// TIA Portal V20 export
// export: Created 2026-04-28T10:05:07.7940218Z, ExportSetting WithDefaults, DisplayName Totally Integrated Automation Portal, DisplayVersion V20, DisplayName TIA Portal Openness, DisplayVersion V20, DisplayName TIA Portal Version Control Interface, DisplayVersion V20, DisplayName SINAMICS Startdrive Advanced, DisplayVersion V20, DisplayName SINAMICS Startdrive G130, G150, S120, S150, SINAMICS MV, G220, S200, S210, DisplayVersion V20, DisplayName SINAMICS Startdrive G110M, G120, G120C, G120D, G120P, G115D, DisplayVersion V20, DisplayName STEP 7 Professional, DisplayVersion V20, DisplayName STEP 7 Safety, DisplayVersion V20, DisplayName WinCC Basic/Comfort/Advanced, DisplayVersion V20, DisplayName WinCC Unified, DisplayVersion V20
TYPE "Daten_SPT_50"
// stored: IsFailsafeCompliant false
   STRUCT
      xMaFa : Bool := false;   // Selection Main fan
      xMaFaSoll : Bool := false;   // Selection Main fan Set Value
      xMaFaIst : Bool := false;   // Selection Main fan Actual Value
      txt_rMoCuMa : DInt := 0;   // Max. motor current, limit
      txt_rMainFanFU : DInt := 0;   // Set Value Main fan
      RangeMainFan : DInt := 0;   // Range Main fan
      xMoCu : Bool := false;   // Selection measurement motor current
      iTakt_MaFa : DInt := 0;   // Interval for recording the measured values
      iAnzWerte_MaFa : DInt := 0;   // Number of measured values
      xFreshAir : Bool := false;   // Selection Fresh air flap
      xComAi : Bool := false;   // Selection Compressed air filter
      xExAir : Bool := false;   // Selection Exhaust air
      xPrCy : Bool := false;   // Selection Pressure in cyclone
      txt_rPrCyMa : DInt := 0;   // Pressure in cyclone Max.
      txt_max_rPrCyMa : DInt := 0;   // Pressure in cyclone Input limit
      RangeCyPr : DInt := 0;   // Range Pressure in cyclone
      iTakt_PrCy : DInt := 0;   // Interval for recording the measured values
      iAnzWerte_PrCy : DInt := 0;   // Number of measured values
      xExAiTe : Bool := false;   // Selection Exhaust air temperature
      txt_rAlExAi : DInt := 0;   // Alarm Exhaust air Valve to open
      txt_rExAiMa : DInt := 0;   // Exhaust air max. Burner off
      txt_rExAiSl : DInt := 0;   // Exhaust air Slip pump on
      txt_rExAiVa : DInt := 0;   // Exhaust air Valve to close
      txt_max_rAlExAi : DInt := 0;   // Exhaust air Valve to close
      txt_max_rExAiMa : DInt := 0;   // Exhaust air max. Burner off
      txt_max_rExAiSl : DInt := 0;   // Exhaust air Slip pump on
      txt_max_rExAiVa : DInt := 0;   // Exhaust air Slip pump on
      xExAirReg : Bool := false;   // Selection with exhaust air control
      txt_rExAiTe : DInt := 0;   // Set Value extract air temperature (control)
      RangeExAi : DInt := 0;   // Range Exhaust air temperature
      iTakt_ExAiTe : DInt := 0;   // Interval for recording the measured values
      iAnzWerte_ExAiTe : DInt := 0;   // Number of measured values
      xFilter : Bool := false;   // Selection filter
      xDiPrFi : Bool := false;   // Selection Differential pressure filter
      txt_rDiPrFiMa : DInt := 0;   // Differential pressure filter Max.
      txt_max_rDiPrFiMa : DInt := 0;   // Differential pressure filter Input Limit
      RangeDiPrFi : DInt := 0;   // Range Differential pressure filter
      iTakt_DiPrFi : DInt := 0;   // Interval for recording the measured values
      iAnzWerte_DiPrFi : DInt := 0;   // Number of measured values
      xDuFiMo : Bool := false;   // Selection Dust filter Monitoring
      txt_rMaxDuFiMo : DInt := 0;   // Dust filter Monitoring Max.
      txt_max_rMaxDuFiMo : DInt := 0;   // Dust filter Monitoring Input Limit
      RangeDuFiMo : DInt := 0;   // Range Dust filter Monitoring
      iTakt_DuFiMo : DInt := 0;   // Interval for recording the measured values
      iAnzWerte_DuFiMo : DInt := 0;   // Number of measured values
      xFlRaAirFlue : Bool := false;   // Selection Volume flow Chimney
      RangeFlRaAirFlue : DInt := 0;   // Range Volume flow Chimney
      xTempFlue : Bool := false;   // Selection Inlet temperature Chimney
      RangeTempFlue : DInt := 0;   // Range Inlet temperature Chimney
      iTakt_FlRaAirFlue : DInt := 0;   // Interval for recording the measured values
      iAnzWerte_FlRaAirFlue : DInt := 0;   // Number of measured values
      iTakt_TempFlue : DInt := 0;   // Interval for recording the measured values
      xPress24_4mA : Bool := false;   // Signal 20-4 ma
      iAnzWerte_TempFlue : DInt := 0;   // Number of measured values
      xVibLimitSw_50 : Bool := 0;   // Selection Dust container fill level
      xHeatExIn : Bool := false;   // Selection Heat exchanger temperature inlet
      RangeHeatExIn : DInt := 0;   // Range Heat exchanger temperature inlet
      iTakt_HeatExIn : DInt := 0;   // Interval for recording the measured values
      iAnzWerte_HeatExIn : DInt := 0;   // Number of measured values
      xHeatExOut : Bool := false;   // Selection Heat exchanger temperature outlet
      RangeHeatExOut : DInt := 0;   // Range Heat exchanger temperature outlet
      iTakt_HeatExOut : DInt := 0;   // Interval for recording the measured values
      iAnzWerte_HeatExOut : DInt := 0;   // Number of measured values
      xDiPrSucFi : Bool := false;   // Selection Differential pressure Filter
      txt_rDiPrSucFiMa : DInt := 0;   // Differential pressure Filter Max.
      txt_max_rDiPrSucFiMa : DInt := 0;   // Differential pressure Filter Input Limit
      RangeDiPrSucFi : DInt := 0;   // Range Differential pressure Filter
      iTakt_DiPrSucFi : DInt := 0;   // Interval for recording the measured values
      iAnzWerte_DiPrSucFi : DInt := 0;   // Number of measured values
      xKnVa50 : Bool := false;   // Selection Knocker valves filter
      t_iKnValve_1 : Time := T#0MS;   // Knocker valves filter On
      t_iKnBreake_1 : Time := T#0MS;   // Knocker valves filter pause
      xOptKnVa : Bool := false;   // Knocker valves automatically
      xOptExAi_min : Bool := false;   // Exhaust air temperature below enable
      txt_rExAi_min : DInt := 0;   // Exhaust air temperature below Min
      xFeedWorm : Bool := false;   // with/without screw conveyor
      x_ExAiTeTB45 : Bool := false;   // Exhaust air monitoring TB45 active 0=no, 1=yes
      x_OptionMitDungsschalter : Bool := false;   // Option With = 1/without =0 Monitoring Dungs switch
      x_OptionMainFanSp : Bool := false;   // Option Main fan with flushing, when starting 0=no, 1=yes
      x_OptionNasswaescher : Bool := false;   // Option Wet washer 0=no, 1=yes
      x_OptionMainFanKlappe : Bool := false;   // Option Exhaust air flaps 0=no, 1=yes
      xFiSysDigital : Bool := false;   // Selection Filter system with digital signals conversion SPT
      xExAiTeCtrl_Intervall : Bool := false;   // Selection Exhaust air temperature monitoring monitoring at defined intervals
      txt_rExAiTeCtrl_Up : DInt := 0;   // Selection Exhaust air temperature monitoring monitoring at defined intervals Up
      txt_rExAiTeCtrl_Down : DInt := 0;   // Selection Exhaust air temperature monitoring monitoring at defined intervals Below
      xOptFiVa : Bool := false;   // Option Filter cleaning valves With = 1 / Without = 0
      t_iFiValve_On : Time := T#0MS;   // Filter cleaning valves With = 1 / Without = 0 Time ON
      t_iFiValveBrake : Time := T#0MS;   // Filter cleaning valves With = 1 / Without = 0 Time break
      xOptPrCompAir : Bool := false;   // Option Compressed Air Sensor Analog With = 1 / Without = 0
      txt_min_rPrCompAir : DInt := 0;   // Compressed Air Min.
      RangePrCompAir : DInt := 0;   // Range Compressed Air Sensor Analog
      iTakt_PrCompAir : DInt := 0;   // Interval for recording the measured values
      iAnzWerte_PrCompAir : DInt := 0;   // Number of measured values
      xOptFlProAir : Bool := false;   // Option Process air quantity With = 1 / Without = 0
      RangeFlProAir : DInt := 0;   // Range Process air quantity With = 1 / Without = 0
      iTakt_FlProAir : DInt := 0;   // Interval for recording the measured values
      iAnzWerte_FlProAir : DInt := 0;   // Number of measured values
      xOptPrFiBefore : Bool := false;   // Option Pressure Filter before With = 1 / Without = 0
      txt_Diff_rPrFi : DInt := 0;   // Difference Pressure Filter before
      RangePrFiBefore : DInt := 0;   // Range Difference Pressure Filter before
      iTakt_PrFiBefore : DInt := 0;   // Interval for recording the measured values
      iAnzWerte_PrFiBefore : DInt := 0;   // Number of measured values
      xOptPrFiAfter : Bool := false;   // Option Pressure Filter after With = 1 / Without = 0
      RangePrFiAfter : DInt := 0;   // Range Difference Pressure Filter after
      iTakt_PrFiAfter : DInt := 0;   // Interval for recording the measured values
      iAnzWerte_PrFiAfter : DInt := 0;   // Number of measured values
      i_AnzahlVentile : DInt := 0;   // Number of valves
      xPrCy_Sensor2 : Bool := false;   // Negative pressure sensor Typ 2 -100 bis 100 mBar Sensortyp 2 = 1
      xOptPrFiBefore_Sensor2 : Bool := false;   // Negative pressure sensor 2 Before
      xOptPrFiAfter_Sensor2 : Bool := false;   // Negative pressure sensor 2 After
      xDiPrFi_AfterFi_S2 : Bool := false;   // Differential pressure with additional sensor after filter Sensor 2 = 1
      txt_rMinProAir : DInt := 0;   // Min. Process Air available
      xTB45EH_Option : Bool := false;   // Option Electric heater TB45 monitoring option 0=No, 1=Yes
      i_TeEH_TB45_Min : DInt := 0;   // Electric heater TB45 monitoring min.
      xDiPrSucFi_S2 : Bool := false;   // Differential pressure with 2 sensors Sensor 2 = 1
      xPrCyCtrl_Intervall : Bool := false;   // Selection Negative pressure Cyclone monitoring at defined intervals
      txt_rPrCyCtrl_Up : DInt := 0;   // Selection Negative pressure Cyclone monitoring at defined intervals Up
      txt_rPrCyCtrl_Down : DInt := 0;   // Selection Negative pressure Cyclone monitoring at defined intervals Below
      xDiPrFiCtrl_Intervall : Bool := false;   // Selection Differential pressure filter monitoring at defined intervals
      txt_rDiPrFiCtrl_Up : DInt := 0;   // Selection Differential pressure filter monitoring at defined intervals Up
      txt_rDiPrFiCtrl_Down : DInt := 0;   // Selection Differential pressure filter monitoring at defined intervals Below
      RangeCyPr_D20 : DInt := 0;   // Range Pressure in cyclone
      txt_rPrCyMa_D20 : DInt := 0;   // Pressure in cyclone Max.
      txt_max_rPrCyMa_D20 : DInt := 0;   // Pressure in cyclone Input limit
      txt_rExAiMa_D20 : DInt := 0;   // Exhaust air max. Burner off
      txt_max_rExAiMa_D20 : DInt := 0;   // Exhaust air max. Burner off Input limit
      RangeExAi_D20 : DInt := 0;   // Range Exhaust air temperature
   END_STRUCT;
END_TYPE
